// TIA Portal V19 export
TYPE "LUC_typeHoldCommandConfiguration"
// Configure in which states a hold command is possible
// stored: Access Published
   STRUCT
      idle : Bool;   // Transition from "Idle" to "Held" is possible
      starting : Bool;   // Transition from "Starting" to "Held" is possible
      suspended : Bool;   // Transition from "Suspended" to "Held" is possible
      execute : Bool := true;   // Transition from "Execute" to "Held" is possible
      unholding : Bool;   // Transition from "Unholding" to "Held" is possible
      suspending : Bool;   // Transition from "Suspending" to "Held" is possible
      unsuspending : Bool;   // Transition from "Unsuspending" to "Held" is possible
      completing : Bool;   // Transition from "Completing" to "Held" is possible
      completed : Bool;   // Transition from "Completed" to "Held" is possible
   END_STRUCT;
END_TYPE
